// TIA Portal V17 export
// export: Created 2026-04-13T11:12:54.5416097Z, ExportSetting WithDefaults, DisplayName Totally Integrated Automation Portal, DisplayVersion V17 Update 4, DisplayName TIA Portal Openness, DisplayVersion V17 Update 4, DisplayName TIA Portal Version Control Interface, DisplayVersion V17, DisplayName SINAMICS Startdrive Advanced, DisplayVersion V17, DisplayName SINAMICS Startdrive G130, G150, S120, S150, SINAMICS MV, S210, DisplayVersion V17, DisplayName SINAMICS Startdrive G110M, G120, G120C, G120D, G120P, G115D, DisplayVersion V17, DisplayName STEP 7 Professional, DisplayVersion V17 Update 4, DisplayName STEP 7 Safety, DisplayVersion V17, DisplayName WinCC Professional, DisplayVersion V17 Update 4
TagTable "BDBS"
  BDBS_SJ事件记录_ : Array [0..19] of String  (PLC tag BDBS.SJ事件记录_, HMI_连接_1, 1 s)
    TagArrayMember "[0]"
    TagArrayMember "[1]"
    TagArrayMember "[2]"
    TagArrayMember "[3]"
    TagArrayMember "[4]"
    TagArrayMember "[5]"
    TagArrayMember "[6]"
    TagArrayMember "[7]"
    TagArrayMember "[8]"
    TagArrayMember "[9]"
    TagArrayMember "[10]"
    TagArrayMember "[11]"
    TagArrayMember "[12]"
    TagArrayMember "[13]"
    TagArrayMember "[14]"
    TagArrayMember "[15]"
    TagArrayMember "[16]"
    TagArrayMember "[17]"
    TagArrayMember "[18]"
    TagArrayMember "[19]"
  BDBS_SJ事件编号 : Array [0..19] of Int  (PLC tag BDBS.SJ事件编号, HMI_连接_1, 1 s)
    TagArrayMember "[0]"
    TagArrayMember "[1]"
    TagArrayMember "[2]"
    TagArrayMember "[3]"
    TagArrayMember "[4]"
    TagArrayMember "[5]"
    TagArrayMember "[6]"
    TagArrayMember "[7]"
    TagArrayMember "[8]"
    TagArrayMember "[9]"
    TagArrayMember "[10]"
    TagArrayMember "[11]"
    TagArrayMember "[12]"
    TagArrayMember "[13]"
    TagArrayMember "[14]"
    TagArrayMember "[15]"
    TagArrayMember "[16]"
    TagArrayMember "[17]"
    TagArrayMember "[18]"
    TagArrayMember "[19]"
  BDBS_QL清零 : Bool  (PLC tag BDBS.QL清零, HMI_连接_1, 1 s)
